# EPICS substitutions: db/user.substitutions
# Example substitutions file

file "db/dbExample1.db" {
    { user = "coudert" }
}

file db/dbExample2.db {
    pattern { user, no, scan }
        { "coudert", 1, "1 second" }
        { "coudert", 2, "2 second" }
        { "coudert", 3, "5 second" }
}
